{attribute addProperty BoxType "EL3004-0000-0020"}
{attribute addProperty Id "AI_Standard_ChannelAT %I*ARRAY[0..3] OF AI_Standard_Channel_F16A160D128160WcStateAT %I*WcState_98A4DF7520.250InfoDataAT %I*InfoData_BC63D37F80100"}
{attribute addProperty CRC "3445512029"}
{attribute addProperty SizeInBites "210"}
{attribute addProperty SizeInBytes "26.25"}
TYPE EL3004_BB821456 :
STRUCT
	{attribute addProperty Name "AI_Standard_Channel"}
	AI_Standard_Channel : ARRAY[0..3] OF AI_Standard_Channel_F16A160D;
	{attribute addProperty Name "WcState"}
	WcState : WcState_98A4DF75;
	{attribute addProperty Name "InfoData"}
	InfoData : InfoData_BC63D37F;
END_STRUCT
END_TYPE

(* stored: Version 1.2.0.0, ProductVersion 3.1.4024.9
   DUT EL3004_BB821456: Id {71ad169c-0596-4752-bd9d-86ef7e26a310} *)
